TYPE ST_MESSAGE_CTRL :
STRUCT
  Cmd         : E_MESSAGE_CTRL;
END_STRUCT
END_TYPE

(* stored: Version 1.1.0.1
   DUT ST_MESSAGE_CTRL: Id {bc46fa2d-a979-4243-8cf0-59a092a9d64c} *)
